{attribute 'qualified_only'}
{attribute 'strict'}
{attribute 'to_string'}
TYPE E_State :
(
	{attribute 'hide'}
	Undefined		:= 0,
	Idle			:= 1,
	
// Start
	Starting		:= 2,
	Execute			:= 3,
	
// Pause
	Pausing			:= 4,
	Paused			:= 5,
	Resuming		:= 6,
	
// Sleep
	Sleeping		:= 7,
	Sleeped			:= 8,

// Stop
	Stopping		:= 9,
	Stopped			:= 10,

// Abort	
	Aborting		:= 11,
	Aborted			:= 12,

// Reset
	Resetting		:= 13

);
END_TYPE

(* stored: Version 1.1.0.1
   DUT E_State: Id {acc0bb97-da91-4632-ac2a-7e54b3136591} *)
